PROGRAM BurningProcess
VAR
	nStep: INT := 0;
END_VAR
VAR_OUTPUT
	err	: UINT;
END_VAR

IF GVL.bBurningStart THEN
	nStep := 1;
	ELSE nStep := 0;
END_IF
CASE nStep OF
	0:
		RETURN;
	1:
		Preparation(nStepIn := nStep, err => GVL.nError, nStepOut => nStep);
		
	2:
		//Ignition(err => GVL.nError);
		//nStep := 0;
	3:
		
END_CASE

END_PROGRAM

(* stored: Version 1.1.0.1, ProductVersion 3.1.4022.18
   POU BurningProcess: Id {c924ffc8-53c3-46d7-8354-936a89d88dbf}, SpecialFunc None *)
